FUNCTION_BLOCK TEST_EQB (* Test EQ function on bit strings *)
  (* Standard: 61499-1 *)
  (* Version 0.0, 2006-09-14, JHC, Holobloc Inc *)
  (* Compiler header: package fb.rt.test; *)
  (* Compiler classdef: SimpleFB *)
  (* Compiler Java Sun JDK 1.5.0 *)
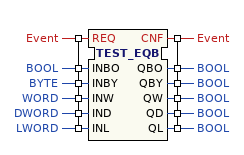
  EVENT_INPUT
    REQ WITH INBO, INBY, INW, IND, INL; (* Normal Execution Request *)
  END_EVENT
  EVENT_OUTPUT
    CNF WITH QBO, QBY, QW, QD, QL; (* Execution Confirmation *)
  END_EVENT
  VAR_INPUT
    INBO : BOOL;
    INBY : BYTE;
    INW : WORD;
    IND : DWORD;
    INL : LWORD;
  END_VAR
  VAR_OUTPUT
    QBO : BOOL;
    QBY : BOOL;
    QW : BOOL;
    QD : BOOL;
    QL : BOOL;
  END_VAR
  ALGORITHM REQ IN FBD:
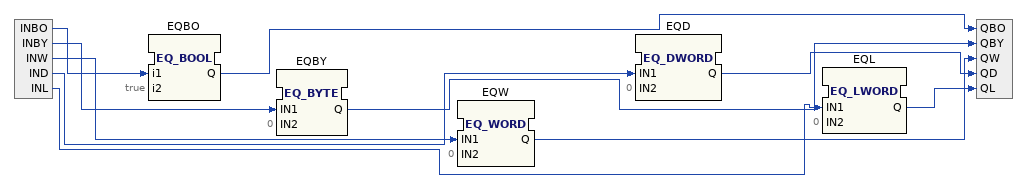
    FBS
      EQBO : EQ_BOOL(i2 := true);
      EQBY : EQ_BYTE(IN2 := 0);
      EQW : EQ_WORD(IN2 := 0);
      EQD : EQ_DWORD(IN2 := 0);
      EQL : EQ_LWORD(IN2 := 0);
    END_FBS
    DATA_CONNECTIONS
      INBO TO EQBO.i1;
      EQBO.Q TO QBO;
      INBY TO EQBY.IN1;
      EQBY.Q TO QBY;
      INW TO EQW.IN1;
      EQW.Q TO QW;
      IND TO EQD.IN1;
      EQD.Q TO QD;
      INL TO EQL.IN1;
      EQL.Q TO QL;
    END_CONNECTIONS
  END_ALGORITHM
END_FUNCTION_BLOCK
